# EPICS IOC start-up script: iocsh/epi8600-meter.iocsh
#- ###         MODBUS   epi8600   iocsh             ###
#- ####################################################
#- >> Mandatory
#- ASYN_PORT_NAME - MODBUS ASYN <name>
#- PREFIX	  - PV PREFIX
#- MODBUS_ADR	  - Modbus address
#- ASLO		  - linear scale for flow rate (0.001
#- 		    for gauge set for Nm³/h, 0.00006
#-		    for gauge set for SLPM
#- SCALE	  - scale factor for total flow
#  		    (1.0 for gauge set for Nm³,
#-		    0.001 for gauge set for SL)
#-
#- >>> Optional
#- KEEP_TCHANGED  - keep the status for the last temperature change
#- 		    (default 900 s). Used for creating sActive status.

#drvModbusAsynConfigure	 'Port name'
#			 'Octet port name'
#			 'Modbus slave address'
#			 'Modbus function code'
#			 'Modbus start address'
#			 'Modbus length'
#			 'Data type'
#			 'Poll time (msec)'
#			 'PLC type'

drvModbusAsynConfigure(RO_DATA_$(ASYN_PORT_NAME)_$(MODBUS_ADR), "$(ASYN_PORT_NAME)", $(MODBUS_ADR), 3, 0x0000, 21, "UINT16", 4000, "epi8600")

drvModbusAsynConfigure(WO_DATA_$(ASYN_PORT_NAME)_$(MODBUS_ADR), "$(ASYN_PORT_NAME)", $(MODBUS_ADR), 16, -1, 2, "UINT16", 0, "epi8600")

#Load your database defining the EPICS records

dbLoadRecords("epi8600.db", "PORT_RO=RO_DATA_$(ASYN_PORT_NAME)_$(MODBUS_ADR),PORT_WO=WO_DATA_$(ASYN_PORT_NAME)_$(MODBUS_ADR),P=$(PREFIX),D=$(DEV_NAME),ASLO=$(ASLO),SCALE=$(SCALE),KEEP_HIGH=$(KEEP_TCHANGED=900.0)")
